(* IEC 61131-3 sources: beckhoffAutomationInterface/ST/Shark/Lib/Hardware/Analog, 5 files *)

(* ---- FB_AnalogInputAdapter.st ---- *)
(*
Generic Analog Channel Adapter for Beckhoff EL3xxx terminals.

Beckhoff auto-generates types with GUID suffixes (e.g., MDP5001_320_5D7E181C) that
change on hardware updates. This adapter uses fixed memory offsets to read channel
data, isolating type dependencies to variable declarations only.

Supported terminals: EL32xx (RTD), EL31xx (voltage/current), EL3174 (pressure)

Memory layout (EL3xxx standard):
Offset 0-1: Status WORD (Underrange=0, Overrange=1, Error=6)
Offset 2-3: Value INT

Usage:
_fbAdapter.Link(pChannel := ADR(_stChannel.MDP5001_xxx_Input));
_fbAdapter.Execute();  // Call each cycle
*)
FUNCTION_BLOCK FB_AnalogInputAdapter IMPLEMENTS I_RawAnalogInput
VAR
    _pChannelData : POINTER TO BYTE;    // Pointer to the hardware channel structure
    _bLinked      : BOOL := FALSE;

    // Cached values (updated in Execute)
    _nRawValue    : DINT;               // 16-bit hardware INT sign-extended to DINT
    _bError       : BOOL;
    _bUnderrange  : BOOL;
    _bOverrange   : BOOL;
END_VAR
VAR CONSTANT
    // Memory offsets for analog channel structure (EL3xxx standard layout)
    OFFSET_STATUS : UINT := 0;          // Status WORD at offset 0
    OFFSET_VALUE  : UINT := 2;          // Value INT at offset 2 (after 2-byte status)

    // Status bit positions (within the 16-bit status word)
    BIT_UNDERRANGE : BYTE := 0;
    BIT_OVERRANGE  : BYTE := 1;
    BIT_ERROR      : BYTE := 6;
END_VAR

    (* Links adapter to the analog channel input structure.
    Pass ADR of the Input member (e.g., ADR(stChannel.MDP5001_xxx_Input)) *)
METHOD PUBLIC Link : BOOL
VAR_INPUT
    pChannel : POINTER TO BYTE;         // Pointer to channel input structure
END_VAR
    IF pChannel = 0 THEN
        _bLinked := FALSE;
        Link := FALSE;
        RETURN;
    END_IF

    _pChannelData := pChannel;
    _bLinked := TRUE;
    Link := TRUE;
END_METHOD

    (* Reads status and value from hardware. Call once per cycle before using GetChannelState. *)
METHOD PUBLIC Execute : BOOL
VAR
    wStatus : WORD;
    pStatus : POINTER TO WORD;
    pValue  : POINTER TO INT;
END_VAR
    IF NOT _bLinked OR _pChannelData = 0 THEN
        _nRawValue := 0;
        _bError := TRUE;
        _bUnderrange := FALSE;
        _bOverrange := FALSE;
        Execute := FALSE;
        RETURN;
    END_IF

    // Read status word from fixed offset
    pStatus := _pChannelData + OFFSET_STATUS;
    wStatus := pStatus^;

    // Extract status bits
    _bUnderrange := (wStatus AND SHL(WORD#1, BIT_UNDERRANGE)) <> 0;
    _bOverrange  := (wStatus AND SHL(WORD#1, BIT_OVERRANGE)) <> 0;
    _bError      := (wStatus AND SHL(WORD#1, BIT_ERROR)) <> 0;

    // Read value from fixed offset (16-bit INT, sign-extended to DINT)
    pValue := _pChannelData + OFFSET_VALUE;
    _nRawValue := INT_TO_DINT(pValue^);

    Execute := TRUE;
END_METHOD

    (* Returns cached channel state. Call Execute() first each cycle. *)
METHOD PUBLIC GetChannelState
VAR_OUTPUT
    nRawValue   : DINT;
    bError      : BOOL;
    bUnderrange : BOOL;
    bOverrange  : BOOL;
END_VAR
    IF _bLinked THEN
        nRawValue   := _nRawValue;
        bError      := _bError;
        bUnderrange := _bUnderrange;
        bOverrange  := _bOverrange;
    ELSE
        nRawValue   := 0;
        bError      := TRUE;
        bUnderrange := FALSE;
        bOverrange  := FALSE;
    END_IF
END_METHOD

    (* Returns TRUE if adapter is linked to hardware. *)
METHOD PUBLIC IsLinked : BOOL
    IsLinked := _bLinked;
END_METHOD

END_FUNCTION_BLOCK

(* ---- FB_AnalogOutput.st ---- *)
(* Analog output control for hardware interface. *)
FUNCTION_BLOCK FB_AnalogOutput IMPLEMENTS I_AnalogOutput
VAR CONSTANT
    MAX_RAW_VALUE : INT := 32767;  // Full scale for 0-10V or 4-20mA outputs
END_VAR
VAR
    _fbError       : FB_ErrorHandler;
    _sInstanceName : STRING(80);
    _Output        : REFERENCE TO INT;
    _nSafeValue    : INT := 0;    // Applied by SetSafeState() — configured at Init time
END_VAR

METHOD PUBLIC Init : BOOL
VAR_INPUT
    sInstanceName : STRING(80);
    ipOutputRef   : REFERENCE TO INT;
    nSafeValue    : INT := 0;     // Raw output value applied when SetSafeState() is called (0 = de-energise)
END_VAR
    _fbError.Init(sInstanceName);
    _sInstanceName := sInstanceName;

    IF NOT __ISVALIDREF(ipOutputRef) THEN
        _fbError.Raise(E_ErrorId.ERR_GEN_NULL_POINTER, 'Output reference is invalid');
        RETURN;
    END_IF

    _Output REF= ipOutputRef;
    _nSafeValue := LIMIT(0, nSafeValue, MAX_RAW_VALUE);
    _fbError.Clear();
    Init := TRUE;
END_METHOD

METHOD PUBLIC SetOutput
VAR_INPUT
    nValue : INT;
END_VAR
    IF __ISVALIDREF(_Output) THEN
        _Output := LIMIT(0, nValue, MAX_RAW_VALUE);
    END_IF
END_METHOD

METHOD PUBLIC SetPercentage
VAR_INPUT
    rPercentage : REAL;
END_VAR
VAR
    rClamped : REAL;
END_VAR
    rClamped := LIMIT(0.0, rPercentage, 100.0);
    SetOutput(REAL_TO_INT(rClamped * INT_TO_REAL(MAX_RAW_VALUE) / 100.0));
END_METHOD

METHOD PUBLIC GetOutput : INT
    IF __ISVALIDREF(_Output) THEN
        GetOutput := _Output;
    END_IF
END_METHOD

METHOD PUBLIC GetPercentage : REAL
    GetPercentage := INT_TO_REAL(GetOutput()) * 100.0 / INT_TO_REAL(MAX_RAW_VALUE);
END_METHOD

METHOD PUBLIC SetSafeState
    IF __ISVALIDREF(_Output) THEN
        _Output := _nSafeValue;
    END_IF
END_METHOD

METHOD PUBLIC GetError : ST_Error
    GetError := _fbError.GetError();
END_METHOD

METHOD PUBLIC IsError : BOOL
    IsError := _fbError.IsActive();
END_METHOD

END_FUNCTION_BLOCK

(* ---- FB_AnalogSensor.st ---- *)
(* Generic analog sensor — reads raw analog input and scales to engineering units.
   Works with any Beckhoff EL3xxx terminal: RTD (EL32xx), current (EL3048/EL3174), voltage (EL31xx).
   Linear mapping: [rawMin, rawMax] → [scaledMin, scaledMax].
   Values outside [scaledMin, scaledMax] are flagged as range errors. *)
FUNCTION_BLOCK FB_AnalogSensor IMPLEMENTS I_Sensor
VAR
    _ipRawInput    : I_RawAnalogInput;
    _rScaledMin    : LREAL;
    _rScaledMax    : LREAL;
    _rScaleFactor  : LREAL;     // Pre-computed: (scaledMax - scaledMin) / (rawMax - rawMin)
    _rOffset       : LREAL;     // Pre-computed: scaledMin - rawMin * scaleFactor
    _bInitialized  : BOOL := FALSE;
    _rCurrentValue : LREAL := 0.0;
    _fbError       : FB_ErrorHandler;
    _fbHwErrTimer  : TON;    // Debounce: fault must persist continuously for HW_ERROR_DEBOUNCE before error is raised
    _rTrigHwErr    : R_TRIG; // Detects rising edge of timer Q — fires once per 5 s period while fault persists
END_VAR

VAR CONSTANT
    HW_ERROR_DEBOUNCE : TIME := T#5S;  // Transient faults shorter than this are silently swallowed
END_VAR

METHOD PUBLIC Init : BOOL
VAR_INPUT
    sInstanceName : STRING(80);
    ipRawInput    : I_RawAnalogInput;
    rRawMin       : LREAL := 0.0;
    rRawMax       : LREAL;
    rScaledMin    : LREAL := 0.0;
    rScaledMax    : LREAL;
END_VAR
    _fbError.Init(sInstanceName);

    IF ipRawInput = 0 THEN
        _fbError.Raise(E_ErrorId.ERR_GEN_NULL_POINTER, 'Null raw input interface');
        RETURN;
    END_IF

    IF rRawMin >= rRawMax THEN
        _fbError.Raise(E_ErrorId.ERR_GEN_INVALID_PARAM, 'Invalid raw range: min >= max');
        RETURN;
    END_IF

    IF rScaledMin >= rScaledMax THEN
        _fbError.Raise(E_ErrorId.ERR_GEN_INVALID_PARAM, 'Invalid scaled range: min >= max');
        RETURN;
    END_IF

    _ipRawInput := ipRawInput;
    _rScaledMin := rScaledMin;
    _rScaledMax := rScaledMax;

    // Pre-compute linear scaling (avoids per-cycle division)
    _rScaleFactor := (rScaledMax - rScaledMin) / (rRawMax - rRawMin);
    _rOffset := rScaledMin - rRawMin * _rScaleFactor;

    _bInitialized := TRUE;
    _fbError.Clear();
    Init := TRUE;
END_METHOD

METHOD PUBLIC Execute : BOOL
VAR
    nRaw        : DINT;
    bErr        : BOOL;
    bUnderrange : BOOL;
    bOverrange  : BOOL;
END_VAR
    IF NOT _bInitialized THEN
        _fbError.Raise(E_ErrorId.ERR_GEN_INITIALIZATION, 'Sensor not initialized');
        RETURN;
    END_IF

    IF _ipRawInput = 0 THEN
        _fbError.Raise(E_ErrorId.ERR_GEN_NULL_POINTER, 'Null raw input interface');
        RETURN;
    END_IF

    _ipRawInput.GetChannelState(nRawValue => nRaw, bError => bErr, bUnderrange => bUnderrange, bOverrange => bOverrange);

    // Always compute the scaled value — even during errors this reflects the actual hardware reading.
    // For overrange (raw=32767) the result lands slightly above rScaledMax, clearly indicating fault.
    // Consumers must call IsError() before trusting the measurement.
    _rCurrentValue := _rOffset + DINT_TO_LREAL(nRaw) * _rScaleFactor;

    // Debounce transient hardware faults: fault must be continuous for HW_ERROR_DEBOUNCE (5 s).
    // After 5 s, _RaiseHwError() is called once. If the fault persists, the timer is immediately
    // reset so it counts another 5 s — giving a periodic log entry every 5 s until the fault clears.
    // R_TRIG detects the Q rising edge so Raise() fires exactly once per 5 s window.
    _fbHwErrTimer(IN := bErr, PT := HW_ERROR_DEBOUNCE);
    _rTrigHwErr(CLK := _fbHwErrTimer.Q);

    IF bErr THEN
        IF _rTrigHwErr.Q THEN
            _RaiseHwError(nRaw, bUnderrange, bOverrange);
            _fbHwErrTimer(IN := FALSE);  // Reset timer: next period starts from 0 on the following cycle
        END_IF
        RETURN;
    END_IF

    IF _fbError.IsActive() THEN
        _fbError.Clear();
    END_IF
    Execute := TRUE;
END_METHOD

// Builds the hardware-error message and raises ERR_HW_SENSOR_OPEN exactly once per fault event.
// Called only on the rising edge of the debounce timer — not on every scan cycle.
METHOD PRIVATE _RaiseHwError
VAR_INPUT
    nRaw        : DINT;
    bUnderrange : BOOL;
    bOverrange  : BOOL;
END_VAR
VAR
    sMsg : STRING(255);
END_VAR
    IF bOverrange THEN
        sMsg := CONCAT('Hardware error - Overrange: raw=', TO_STRING(nRaw));
    ELSIF bUnderrange THEN
        sMsg := CONCAT('Hardware error - Underrange: raw=', TO_STRING(nRaw));
    ELSE
        sMsg := 'Hardware error';
    END_IF
    _fbError.Clear();  // Reset dedup guard so Raise() logs every periodic re-raise, not just the first
    _fbError.Raise(E_ErrorId.ERR_HW_SENSOR_OPEN, sMsg);
END_METHOD

// -----------------------------------------------------------------------------
// I_Sensor
// -----------------------------------------------------------------------------
METHOD PUBLIC GetMeasurement : LREAL
    GetMeasurement := _rCurrentValue;
END_METHOD

// -----------------------------------------------------------------------------
// I_Errorable
// -----------------------------------------------------------------------------
METHOD PUBLIC IsError : BOOL
    IsError := _fbError.IsActive();
END_METHOD

METHOD PUBLIC GetError : ST_Error
    GetError := _fbError.GetError();
END_METHOD

END_FUNCTION_BLOCK

(* ---- FB_DualSensor.st ---- *)
(* Dual sensor composite — averages two I_Sensor readings with deviation monitoring. *)
FUNCTION_BLOCK FB_DualSensor IMPLEMENTS I_Sensor

VAR
    // Sensor references
    _ipPrimarySensor    : I_Sensor;
    _ipSecondarySensor  : I_Sensor;

    // Configuration
    _rMaxDeviation      : LREAL := 5.0;          // Max allowed sensor difference

    // State
    _bInitialized       : BOOL := FALSE;
    _bUseDualSensors    : BOOL := FALSE;
    _rCurrentValue      : LREAL := 0.0;          // Current averaged value
    _rDeviation         : LREAL := 0.0;          // Sensor deviation (dual mode only)
    _fbError            : FB_ErrorHandler;       // Centralized error handling
END_VAR

METHOD PUBLIC Init : BOOL
VAR_INPUT
    sInstanceName       : STRING(80);            // Instance name for error source
    ipPrimary           : I_Sensor;              // Primary sensor (required)
    ipSecondary         : I_Sensor;              // Secondary sensor (optional, 0 = single mode)
    rMaxDeviation       : LREAL := 5.0;          // Max sensor deviation
END_VAR
    _fbError.Init(sInstanceName);

    IF ipPrimary = 0 THEN
        _fbError.Raise(E_ErrorId.ERR_GEN_NULL_POINTER, 'Primary sensor reference is null');
        RETURN;
    END_IF

    _ipPrimarySensor := ipPrimary;
    _ipSecondarySensor := ipSecondary;
    _rMaxDeviation := rMaxDeviation;

    _bUseDualSensors := (ipSecondary <> 0);
    _bInitialized := TRUE;
    _fbError.Clear();

    Init := TRUE;
END_METHOD

METHOD PUBLIC Execute : BOOL
VAR
    rPrimary      : LREAL;
    rSecondary    : LREAL;
END_VAR

    Execute := FALSE;

    // 1. Initialization Check
    IF NOT _bInitialized THEN
        _fbError.Raise(E_ErrorId.ERR_GEN_INITIALIZATION, 'Dual sensor not initialized');
        RETURN;
    END_IF

    // 2. Primary Sensor Check - Preserve child error details
    IF _ipPrimarySensor.IsError() THEN
        _fbError.RaiseFromChild(_ipPrimarySensor.GetError());
        RETURN;
    END_IF
    rPrimary := _ipPrimarySensor.GetMeasurement();

    // 3. Single Sensor Mode (Early Exit)
    IF NOT _bUseDualSensors THEN
        _rCurrentValue := rPrimary;
        _rDeviation := 0.0;
        IF _fbError.IsActive() THEN
            _fbError.Clear();
        END_IF
        Execute := TRUE;
        RETURN;
    END_IF

    // 4. Secondary Sensor Check - Preserve child error details
    IF _ipSecondarySensor.IsError() THEN
        _fbError.RaiseFromChild(_ipSecondarySensor.GetError());
        RETURN;
    END_IF
    rSecondary := _ipSecondarySensor.GetMeasurement();

    // 5. Calculate average regardless of deviation check
    _rCurrentValue := (rPrimary + rSecondary) / 2.0;

    // 6. Deviation Check - include actual values in message
    _rDeviation := ABS(rPrimary - rSecondary);

    IF _rDeviation > _rMaxDeviation THEN
        _fbError.RaiseWithValues(E_ErrorId.ERR_CTRL_DEVIATION_HIGH, 'Deviation', _rDeviation, _rMaxDeviation, '');
        RETURN;
    END_IF

    // 7. Success
    IF _fbError.IsActive() THEN
        _fbError.Clear();
    END_IF
    Execute := TRUE;
END_METHOD

METHOD PUBLIC GetDeviation : LREAL
    GetDeviation := _rDeviation;
END_METHOD

METHOD PUBLIC IsDualSensor : BOOL
    IsDualSensor := _bUseDualSensors;
END_METHOD

METHOD PUBLIC GetMeasurement : LREAL
    GetMeasurement := _rCurrentValue;
END_METHOD

METHOD PUBLIC IsError : BOOL
    IsError := _fbError.IsActive();
END_METHOD

METHOD PUBLIC GetError : ST_Error
    GetError := _fbError.GetError();
END_METHOD

END_FUNCTION_BLOCK

(* ---- FB_TcInputAdapter.st ---- *)
(*
EL3314 Thermocouple Channel Adapter for Beckhoff EL3314-xxxx terminals.

Beckhoff auto-generates types with GUID suffixes (e.g., MDP5001_330_88CAB57D) that
change on hardware updates. This adapter uses fixed memory offsets to read channel
data, isolating type dependencies to variable declarations only.

Unlike FB_AnalogInputAdapter (16-bit INT value at offset 2), the EL3314 channel
PDO carries a 32-bit DINT value preceded by a reserved word:

Memory layout (EL3314 channel, MDP5001_330_C_I_D7C99110):
Offset 0-1: Status WORD (Underrange=0, Overrange=1, Error=6)
Offset 2-3: _reserved UINT
Offset 4-7: Value DINT

Usage:
_fbAdapter.Link(pChannel := ADR(_stTerminal.In.TC_Inputs_Channel_1));
_fbAdapter.Execute();  // Call each cycle
*)
FUNCTION_BLOCK FB_TcInputAdapter IMPLEMENTS I_RawAnalogInput
VAR
    _pChannelData : POINTER TO BYTE;    // Pointer to the hardware channel structure
    _bLinked      : BOOL := FALSE;

    // Cached values (updated in Execute)
    _nRawValue    : DINT;               // 32-bit thermocouple counts
    _bError       : BOOL;
    _bUnderrange  : BOOL;
    _bOverrange   : BOOL;
END_VAR
VAR CONSTANT
    // Memory offsets for EL3314 channel structure
    OFFSET_STATUS : UINT := 0;          // Status WORD at offset 0
    OFFSET_VALUE  : UINT := 4;          // Value DINT at offset 4 (after status + reserved word)

    // Status bit positions (within the 16-bit status word)
    BIT_UNDERRANGE : BYTE := 0;
    BIT_OVERRANGE  : BYTE := 1;
    BIT_ERROR      : BYTE := 6;
END_VAR

    (* Links adapter to the thermocouple channel input structure.
    Pass ADR of the channel member (e.g., ADR(stTerminal.In.TC_Inputs_Channel_1)) *)
METHOD PUBLIC Link : BOOL
VAR_INPUT
    pChannel : POINTER TO BYTE;         // Pointer to channel input structure
END_VAR
    IF pChannel = 0 THEN
        _bLinked := FALSE;
        Link := FALSE;
        RETURN;
    END_IF

    _pChannelData := pChannel;
    _bLinked := TRUE;
    Link := TRUE;
END_METHOD

    (* Reads status and value from hardware. Call once per cycle before using GetChannelState. *)
METHOD PUBLIC Execute : BOOL
VAR
    wStatus : WORD;
    pStatus : POINTER TO WORD;
    pValue  : POINTER TO DINT;
END_VAR
    IF NOT _bLinked OR _pChannelData = 0 THEN
        _nRawValue := 0;
        _bError := TRUE;
        _bUnderrange := FALSE;
        _bOverrange := FALSE;
        Execute := FALSE;
        RETURN;
    END_IF

    // Read status word from fixed offset
    pStatus := _pChannelData + OFFSET_STATUS;
    wStatus := pStatus^;

    // Extract status bits
    _bUnderrange := (wStatus AND SHL(WORD#1, BIT_UNDERRANGE)) <> 0;
    _bOverrange  := (wStatus AND SHL(WORD#1, BIT_OVERRANGE)) <> 0;
    _bError      := (wStatus AND SHL(WORD#1, BIT_ERROR)) <> 0;

    // Read 32-bit value from fixed offset
    pValue := _pChannelData + OFFSET_VALUE;
    _nRawValue := pValue^;

    Execute := TRUE;
END_METHOD

    (* Returns cached channel state. Call Execute() first each cycle. *)
METHOD PUBLIC GetChannelState
VAR_OUTPUT
    nRawValue   : DINT;
    bError      : BOOL;
    bUnderrange : BOOL;
    bOverrange  : BOOL;
END_VAR
    IF _bLinked THEN
        nRawValue   := _nRawValue;
        bError      := _bError;
        bUnderrange := _bUnderrange;
        bOverrange  := _bOverrange;
    ELSE
        nRawValue   := 0;
        bError      := TRUE;
        bUnderrange := FALSE;
        bOverrange  := FALSE;
    END_IF
END_METHOD

    (* Returns TRUE if adapter is linked to hardware. *)
METHOD PUBLIC IsLinked : BOOL
    IsLinked := _bLinked;
END_METHOD

END_FUNCTION_BLOCK
